PROGRAM zadanie_zapocet
VAR
	M1: BOOL;
	M2: BOOL;
	M3: BOOL;
	start: BOOL;
	stop1: BOOL;
	stav: UINT;
	stop2: BOOL;
	stop3: BOOL;
	casovac: TON;
END_VAR

CASE stav OF 
	0: M1 := FALSE; 
	   M2 := FALSE; 
	   M3 := FALSE; 
	   casovac.IN := FALSE; 
	   casovac(); 
	IF start = TRUE THEN
		stav := 10; 
	END_IF
	10: M1 := TRUE; 
		M2 := FALSE; 
		M3 := FALSE; 
		casovac.IN := TRUE; 
		casovac.PT := T#5S; 
		casovac(); 
		IF casovac.Q = TRUE THEN
			stav := 20; 
		END_IF
		
	20: M1 := TRUE;
		M2 := TRUE;
		M3 := TRUE;
	IF stop1 = TRUE THEN 
		stav := 30;
		END_IF
	30: M1 := FALSE;
		M2 := TRUE;
		M3 := TRUE;
	IF stop3 = TRUE THEN 
		stav := 40;
	END_IF
	40: M1 := FALSE;
		M2 := TRUE;
		M3 := FALSE;
	IF stop2 = TRUE THEN 
		stav := 50;
	END_IF
	50: M1 := FALSE;
		M2 := FALSE;
		M3 := FALSE;
END_CASE

END_PROGRAM

(* stored: Version 1.1.0.1, ProductVersion 3.1.4024.16
   POU zadanie_zapocet: Id {ee0566a5-4229-4650-8504-ee09e0a8567d}, SpecialFunc None *)
